// TIA Portal V20 export
FUNCTION_BLOCK "AdjLeft"   // FB525, FBD
{ S7_Optimized_Access := 'TRUE' }
// stored: AutoNumber false, MemoryReserve 100, SetENOAutomatically false
   VAR
      Var { ExternalAccessible := 'False'; ExternalVisible := 'False'; ExternalWritable := 'False'} : "TypeVar";
      Cmd { ExternalAccessible := 'False'; ExternalVisible := 'False'; ExternalWritable := 'False'} : "TypeCmd";
      Enc { ExternalAccessible := 'False'; ExternalVisible := 'False'; ExternalWritable := 'False'} : "SysCounterFast";
      Pos { ExternalAccessible := 'False'; ExternalVisible := 'False'; ExternalWritable := 'False'} : "SysPos";
      AdjSlow { ExternalAccessible := 'False'; ExternalVisible := 'False'; ExternalWritable := 'False'} : "SysMotor";
      AdjFast { ExternalAccessible := 'False'; ExternalVisible := 'False'; ExternalWritable := 'False'} : "SysLinMotC1150";
      TAutoOn { ExternalAccessible := 'False'; ExternalVisible := 'False'; ExternalWritable := 'False'} : TON_TIME;
      TAutoTarPosManOn { ExternalAccessible := 'False'; ExternalVisible := 'False'; ExternalWritable := 'False'} : TON_TIME;
      T { ExternalAccessible := 'False'; ExternalVisible := 'False'; ExternalWritable := 'False'} : Array[1..5] of IEC_TIMER;
      adjFastPnSlaveOff { ExternalAccessible := 'False'; ExternalVisible := 'False'; ExternalWritable := 'False'} : "SysPnSlaveDeactivate";
      tarOld { ExternalAccessible := 'False'; ExternalVisible := 'False'; ExternalWritable := 'False'} : DInt;
      autoTarPosMan { ExternalAccessible := 'False'; ExternalVisible := 'False'; ExternalWritable := 'False'} : Bool;
      setValueEnc { ExternalAccessible := 'False'; ExternalVisible := 'False'; ExternalWritable := 'False'} : Bool;
      autoRef { ExternalAccessible := 'False'; ExternalVisible := 'False'; ExternalWritable := 'False'} : Bool;
      posOld { ExternalAccessible := 'False'; ExternalVisible := 'False'; ExternalWritable := 'False'} : Real;
      posDiff { ExternalAccessible := 'False'; ExternalVisible := 'False'; ExternalWritable := 'False'} : Real;
   END_VAR
   VAR_TEMP
      CtrlPc : Struct
         ackErr : Bool;
         manModeActive : Bool;
         manP : Bool;
         manM : Bool;
         manRefRun : Bool;
      END_STRUCT;
      CtrlLinMot : Struct
         mode : Int;
         target : Real;
         acc : Real;
         dec : Real;
         jerk : Real;
         speed : Real;
      END_STRUCT;
      refPosDiff : DInt;
      offsetNoStd : Real;
      refPosDiffCalib : DInt;
      modeCalib : Int;
      disMechanicToZero : Int;   // distance mechanic part left to zero [mm]
   END_VAR
   VAR_TEMP   // added for the SCL form of the ladder/FBD networks
      _w1 : Bool;
   END_VAR
BEGIN

REGION Network 1 (SCL): offset for no standard calibration
   (* 
   normally the distance from camera TO board should be 550mm
   for special application the distance is different
   the distance can be changed in the goldeneye program
   if its different then 550mm a offset will be added
   *)
   #offsetNoStd := 0.0;
   IF "ComRd".Data.Left.RefPosToBoard <> 550 THEN
       #offsetNoStd := (DINT_TO_REAL("ComRd".Data.Left.RefPosToBoard) - 550.0);
   ELSE
       #offsetNoStd := 0.0;
   END_IF;
END_REGION

REGION Network 2 (SCL): calibration value for offset
   (* 
   modus for calibartion
   camera must be referenced first
   mode 1 -->   the camera must be moved manually to position 550mm from board and
                 then press "Set Nullpoint"
   mode 2 -->   the camera must be moved to a other position and
                 then must be measured from the calibration tool to the camera and
                 this value must be putted in after pressing "Set Nullpoint"
   *)     
   #disMechanicToZero := 870;  
   #modeCalib := 2;
   IF #modeCalib = 1 THEN
       #refPosDiffCalib := "ComRd".Data.Left.TargetPos;
   ELSIF #modeCalib = 2 THEN
       #refPosDiffCalib := (#disMechanicToZero * 10) - ("ComRd".Data.Left.CalibratePos + 5500);
   END_IF;
END_REGION

REGION Network 3 (SCL): calibration value from pc
   "ComSd".Data.Left.SetCalibratePosOk := FALSE;

   IF "ComRd".Data.Left.SetCalibratePos THEN

       IF "G".Cfg.adjLeftActive THEN
           #refPosDiff := REAL_TO_DINT("Enc"."8BC1.L".act * 10.0) - #refPosDiffCalib;
       ELSIF "G".Cfg.adjLeftActiveLinMot THEN
           #refPosDiff := REAL_TO_DINT("Enc"."8U1.L".act * 10.0) - #refPosDiffCalib;
       END_IF;

       "Ref".adjLeftCalOffset := #refPosDiff;
       "ComSd".Data.Left.SetCalibratePosOk := TRUE;

   END_IF;
END_REGION

REGION Network 4 (SCL): target position
   #Cmd.target := "G".Batch.width / 2.0;
   IF "G".Cfg.modeBoardPassing = 2 AND ("G".Cfg.modeDimension = 2 OR "G".Cfg.modeDimension = 4) AND NOT "G".Batch.stdActive THEN
       #Cmd.target := "G".Batch.width / 2.0 + ("G".Batch.widthMeasure - "G".Batch.width);
   END_IF;

   IF "G".Cfg.modeBoardPassing = 3 AND ("G".Cfg.modeDimension = 2 OR "G".Cfg.modeDimension = 4) AND NOT "G".Batch.stdActive THEN
       #Cmd.target := "G".Batch.senLeftVal;
   END_IF;

   IF #autoTarPosMan THEN
       #Cmd.target := DINT_TO_REAL(("ComRd".Data.Left.TargetPos)) / 10.0;
   END_IF;

   "Ref".adjLeftTar := #Cmd.target + (DINT_TO_REAL("Ref".adjLeftCalOffset) / 10.0) + #offsetNoStd + "Enc"."8B1.B".offset;
END_REGION

REGION Network 5 (SCL): data from pc
   IF NOT "G".errComPc THEN
       #CtrlPc.manModeActive := "ComRd".Data.Left.ManModeActive;
       #CtrlPc.manP := "ComRd".Data.Left.ManPlus;
       #CtrlPc.manM := "ComRd".Data.Left.ManMinus;
       #CtrlPc.manRefRun := "ComRd".Data.Left.ManRefRun;
   ELSE
       #CtrlPc.manModeActive := TRUE;
       #CtrlPc.manP := FALSE;
       #CtrlPc.manM := FALSE;
       #CtrlPc.manRefRun := FALSE;
   END_IF;
   #CtrlPc.ackErr := "G".ack;
END_REGION

REGION Network 6: off
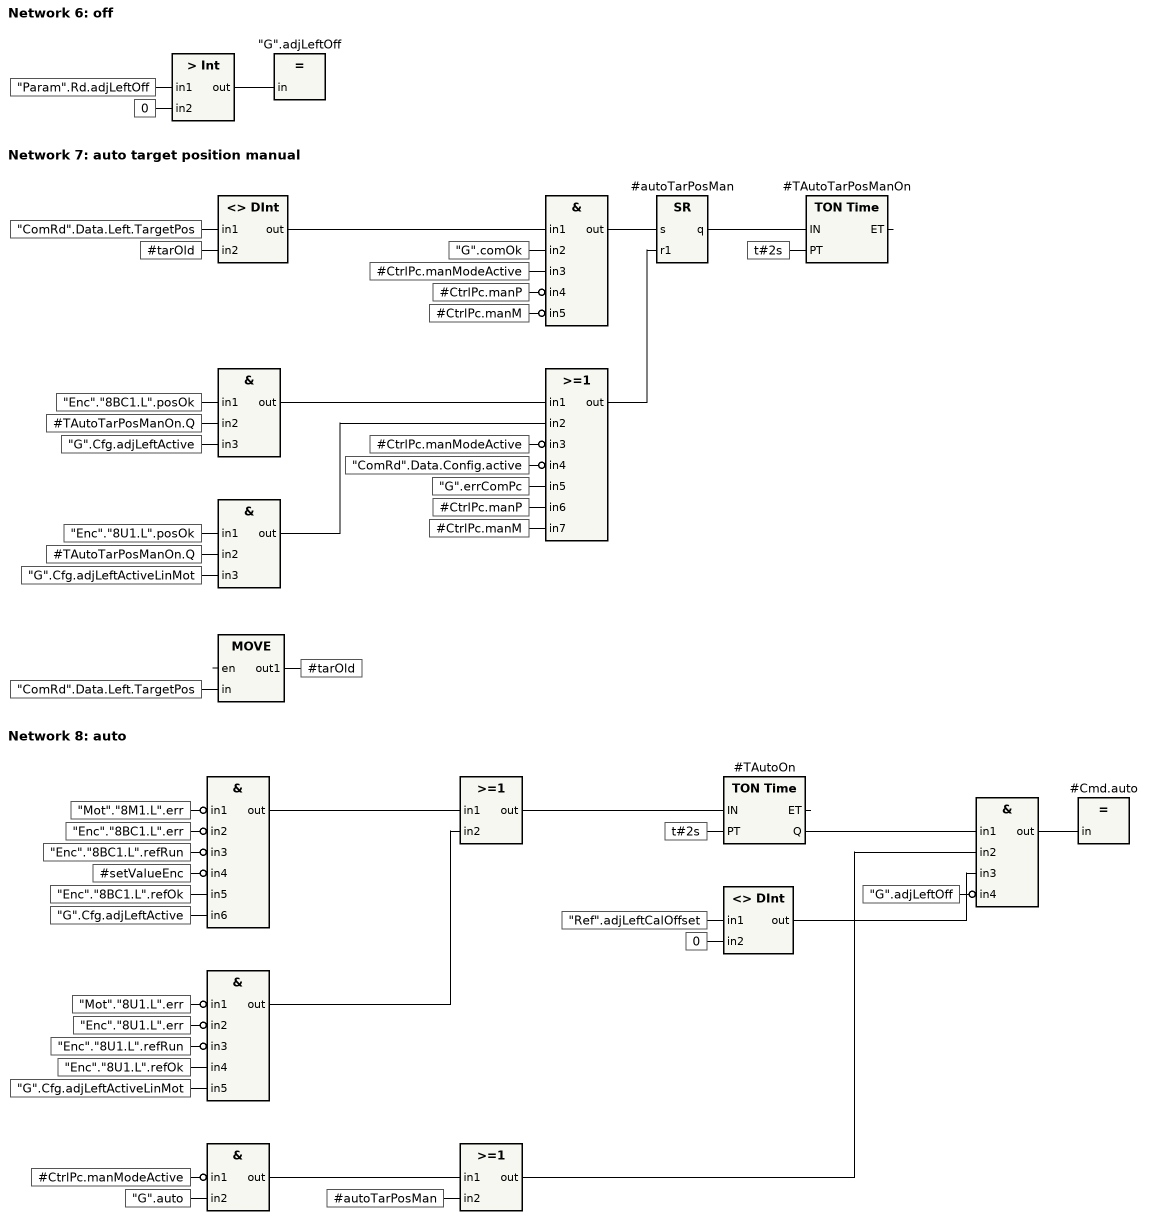
   "G".adjLeftOff := "Param".Rd.adjLeftOff > 0;
END_REGION

REGION Network 7: auto target position manual
   IF ("ComRd".Data.Left.TargetPos <> #tarOld) AND "G".comOk AND #CtrlPc.manModeActive AND NOT #CtrlPc.manP AND NOT #CtrlPc.manM THEN
       #autoTarPosMan := TRUE;   // SR flip-flop
   END_IF;
   IF ("Enc"."8BC1.L".posOk AND #TAutoTarPosManOn.Q AND "G".Cfg.adjLeftActive) OR ("Enc"."8U1.L".posOk AND #TAutoTarPosManOn.Q AND "G".Cfg.adjLeftActiveLinMot) OR NOT #CtrlPc.manModeActive OR NOT "ComRd".Data.Config.active OR "G".errComPc OR #CtrlPc.manP OR #CtrlPc.manM THEN
       #autoTarPosMan := FALSE;
   END_IF;
   #TAutoTarPosManOn(IN := #autoTarPosMan, PT := t#2s);   // TON
   #tarOld := "ComRd".Data.Left.TargetPos;
END_REGION

REGION Network 8: auto
   #TAutoOn(IN := (NOT "Mot"."8M1.L".err AND NOT "Enc"."8BC1.L".err AND NOT "Enc"."8BC1.L".refRun AND NOT #setValueEnc AND "Enc"."8BC1.L".refOk AND "G".Cfg.adjLeftActive) OR (NOT "Mot"."8U1.L".err AND NOT "Enc"."8U1.L".err AND NOT "Enc"."8U1.L".refRun AND "Enc"."8U1.L".refOk AND "G".Cfg.adjLeftActiveLinMot),   // TON
            PT := t#2s);
   #Cmd.auto := #TAutoOn.Q AND ((NOT #CtrlPc.manModeActive AND "G".auto) OR #autoTarPosMan) AND ("Ref".adjLeftCalOffset <> 0) AND NOT "G".adjLeftOff;
END_REGION

REGION Network 9: manual
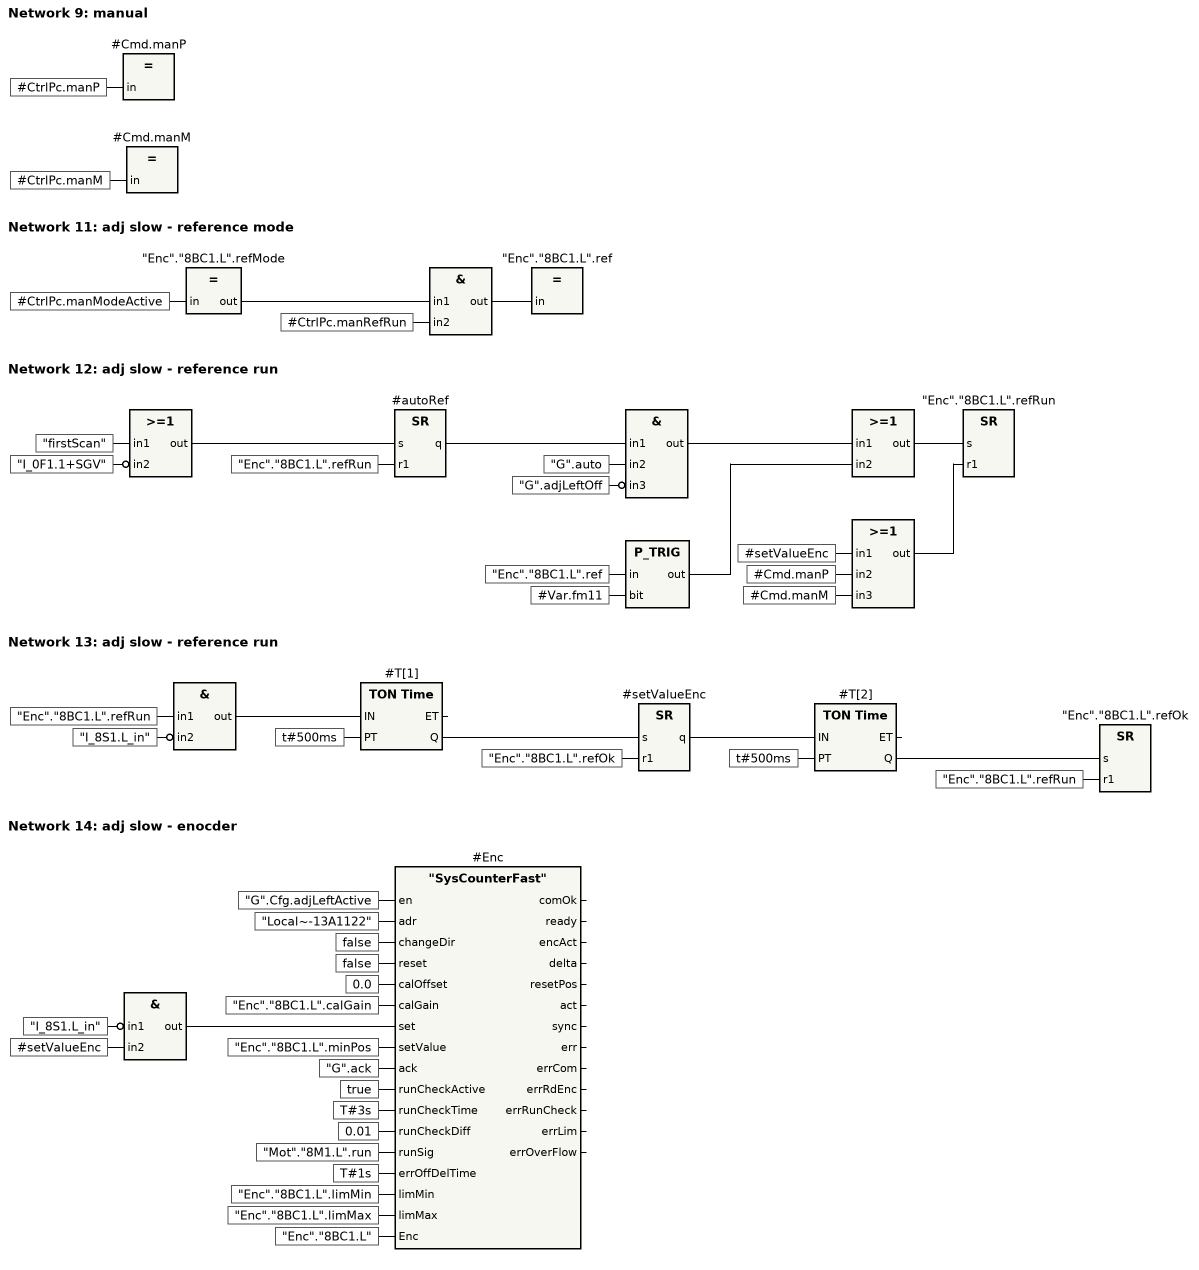
   #Cmd.manP := #CtrlPc.manP;
   #Cmd.manM := #CtrlPc.manM;
END_REGION

REGION Network 10 (SCL): adj slow - calibration value
   "Enc"."8BC1.L".calGain := -0.0275;

   "Enc"."8BC1.L".minPos := 10.0;
   "Enc"."8BC1.L".maxPos := 210.0;

   "Enc"."8BC1.L".limMin := "Enc"."8BC1.L".minPos - 5.0;
   "Enc"."8BC1.L".limMax := "Enc"."8BC1.L".maxPos + 5.0;

   "Enc"."8BC1.L".tarMinPos := "Enc"."8BC1.L".minPos + 0.0;
   "Enc"."8BC1.L".tarMaxPos := "Enc"."8BC1.L".maxPos - 0.0;
END_REGION

REGION Network 11: adj slow - reference mode
   "Enc"."8BC1.L".refMode := #CtrlPc.manModeActive;
   "Enc"."8BC1.L".ref := #CtrlPc.manModeActive AND #CtrlPc.manRefRun;
END_REGION

REGION Network 12: adj slow - reference run
   IF "firstScan" OR NOT "I_0F1.1+SGV" THEN
       #autoRef := TRUE;   // SR flip-flop
   END_IF;
   IF "Enc"."8BC1.L".refRun THEN #autoRef := FALSE; END_IF;
   #_w1 := "Enc"."8BC1.L".ref AND NOT #Var.fm11;   // rising edge
   #Var.fm11 := "Enc"."8BC1.L".ref;
   IF (#autoRef AND "G".auto AND NOT "G".adjLeftOff) OR #_w1 THEN
       "Enc"."8BC1.L".refRun := TRUE;   // SR flip-flop
   END_IF;
   IF #setValueEnc OR #Cmd.manP OR #Cmd.manM THEN "Enc"."8BC1.L".refRun := FALSE; END_IF;
END_REGION

REGION Network 13: adj slow - reference run
   #T[1].TON(IN := "Enc"."8BC1.L".refRun AND NOT "I_8S1.L_in", PT := t#500ms);
   IF #T[1].Q THEN
       #setValueEnc := TRUE;   // SR flip-flop
   END_IF;
   IF "Enc"."8BC1.L".refOk THEN #setValueEnc := FALSE; END_IF;
   #T[2].TON(IN := #setValueEnc, PT := t#500ms);
   IF #T[2].Q THEN
       "Enc"."8BC1.L".refOk := TRUE;   // SR flip-flop
   END_IF;
   IF "Enc"."8BC1.L".refRun THEN "Enc"."8BC1.L".refOk := FALSE; END_IF;
END_REGION

REGION Network 14: adj slow - enocder
   IF "G".Cfg.adjLeftActive THEN
       #Enc(adr := "Local~-13A1122",   // "SysCounterFast"
            changeDir := false,
            reset := false,
            calOffset := 0.0,
            calGain := "Enc"."8BC1.L".calGain,
            set := NOT "I_8S1.L_in" AND #setValueEnc,
            setValue := "Enc"."8BC1.L".minPos,
            ack := "G".ack,
            runCheckActive := true,
            runCheckTime := T#3s,
            runCheckDiff := 0.01,
            runSig := "Mot"."8M1.L".run,
            errOffDelTime := T#1s,
            limMin := "Enc"."8BC1.L".limMin,
            limMax := "Enc"."8BC1.L".limMax,
            Enc := "Enc"."8BC1.L");
   END_IF;
END_REGION

REGION Network 15: adj slow - pos
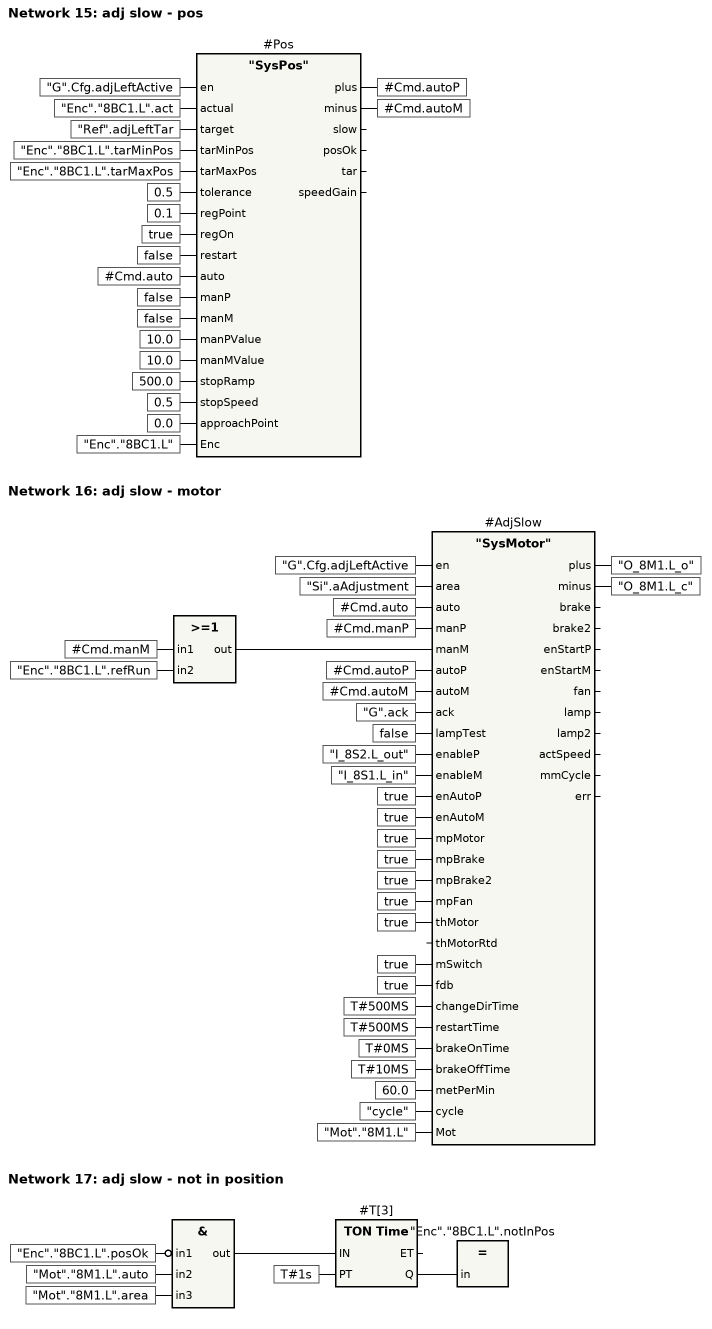
   IF "G".Cfg.adjLeftActive THEN
       #Pos(actual := "Enc"."8BC1.L".act,   // "SysPos"
            target := "Ref".adjLeftTar,
            tarMinPos := "Enc"."8BC1.L".tarMinPos,
            tarMaxPos := "Enc"."8BC1.L".tarMaxPos,
            tolerance := 0.5,
            regPoint := 0.1,
            regOn := true,
            restart := false,
            auto := #Cmd.auto,
            manP := false,
            manM := false,
            manPValue := 10.0,
            manMValue := 10.0,
            stopRamp := 500.0,
            stopSpeed := 0.5,
            approachPoint := 0.0,
            Enc := "Enc"."8BC1.L",
            plus => #Cmd.autoP,
            minus => #Cmd.autoM);
   END_IF;
END_REGION

REGION Network 16: adj slow - motor
   IF "G".Cfg.adjLeftActive THEN
       #AdjSlow(area := "Si".aAdjustment,   // "SysMotor"
                auto := #Cmd.auto,
                manP := #Cmd.manP,
                manM := #Cmd.manM OR "Enc"."8BC1.L".refRun,
                autoP := #Cmd.autoP,
                autoM := #Cmd.autoM,
                ack := "G".ack,
                lampTest := false,
                enableP := "I_8S2.L_out",
                enableM := "I_8S1.L_in",
                enAutoP := true,
                enAutoM := true,
                mpMotor := true,
                mpBrake := true,
                mpBrake2 := true,
                mpFan := true,
                thMotor := true,
                mSwitch := true,
                fdb := true,
                changeDirTime := T#500MS,
                restartTime := T#500MS,
                brakeOnTime := T#0MS,
                brakeOffTime := T#10MS,
                metPerMin := 60.0,
                cycle := "cycle",
                Mot := "Mot"."8M1.L",
                plus => "O_8M1.L_o",
                minus => "O_8M1.L_c");
   END_IF;
END_REGION

REGION Network 17: adj slow - not in position
   #T[3].TON(IN := NOT "Enc"."8BC1.L".posOk AND "Mot"."8M1.L".auto AND "Mot"."8M1.L".area, PT := T#1s);
   "Enc"."8BC1.L".notInPos := #T[3].Q;
END_REGION

REGION Network 18: adj slow - sensor monitoring
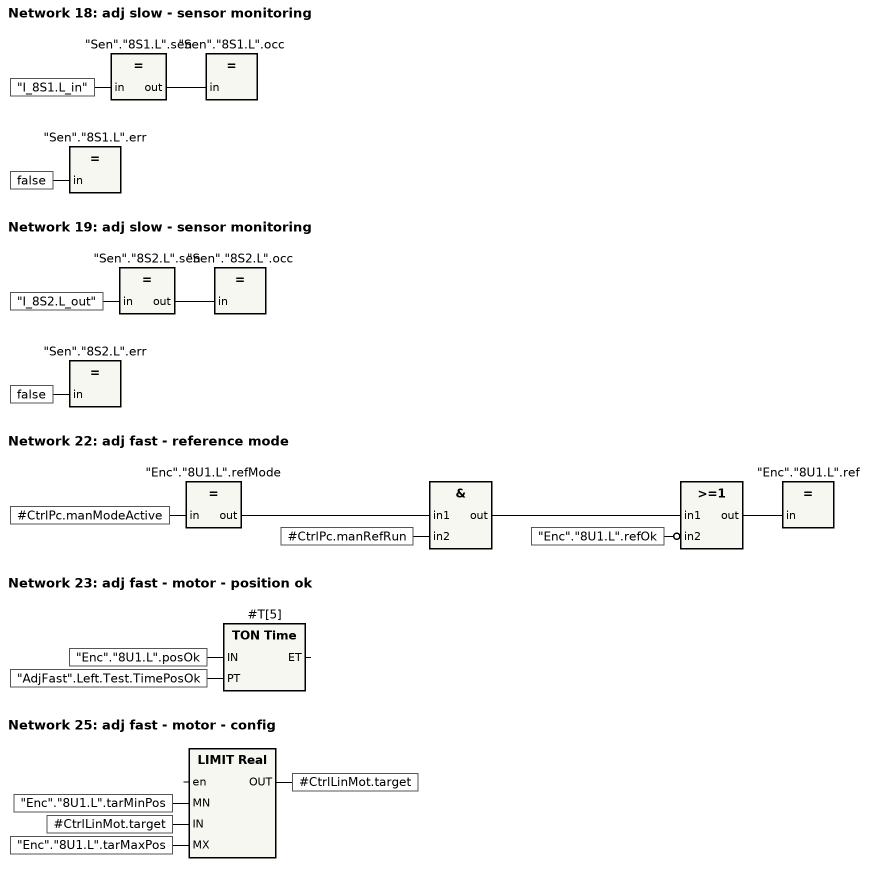
   "Sen"."8S1.L".sen := "I_8S1.L_in";
   "Sen"."8S1.L".occ := "I_8S1.L_in";
   "Sen"."8S1.L".err := false;
END_REGION

REGION Network 19: adj slow - sensor monitoring
   "Sen"."8S2.L".sen := "I_8S2.L_out";
   "Sen"."8S2.L".occ := "I_8S2.L_out";
   "Sen"."8S2.L".err := false;
END_REGION

REGION Network 21 (SCL): adj fast - calibration value
   "Enc"."8U1.L".calGain := 1.0;

   "Enc"."8U1.L".minPos := 5.0;
   "Enc"."8U1.L".maxPos := 155.0;

   "Enc"."8U1.L".limMin := "Enc"."8U1.L".minPos - 5.0;
   "Enc"."8U1.L".limMax := "Enc"."8U1.L".maxPos + 5.0;

   "Enc"."8U1.L".tarMinPos := "Enc"."8U1.L".minPos + 0.0;
   "Enc"."8U1.L".tarMaxPos := "Enc"."8U1.L".maxPos - 0.0;
END_REGION

REGION Network 22: adj fast - reference mode
   "Enc"."8U1.L".refMode := #CtrlPc.manModeActive;
   "Enc"."8U1.L".ref := (#CtrlPc.manModeActive AND #CtrlPc.manRefRun) OR NOT "Enc"."8U1.L".refOk;
END_REGION

REGION Network 23: adj fast - motor - position ok
   #T[5].TON(IN := "Enc"."8U1.L".posOk, PT := "AdjFast".Left.Test.TimePosOk);
END_REGION

REGION Network 24 (SCL): adj fast - motor - config

   //############################################################
   // min            5     mm
   // max          155     mm

   // speed        02      m/s
   // acc/dec      24      m/s2
   // jerk         450     m/s3

   // mode         BestehornVAJ
   //############################################################

   // only testmode for plc
   IF "AdjFast".Left.Test.ModeActive AND NOT #CtrlPc.manModeActive THEN
       IF "AdjFast".Left.Test.TarPos = "AdjFast".Left.Test.TarPos1 AND #T[5].Q THEN
           "AdjFast".Left.Test.TarPos := "AdjFast".Left.Test.TarPos2;
       ELSIF "AdjFast".Left.Test.TarPos = "AdjFast".Left.Test.TarPos2 AND #T[5].Q THEN
           "AdjFast".Left.Test.TarPos := "AdjFast".Left.Test.TarPos1;
       END_IF;
       "Ref".adjLeftTar := "AdjFast".Left.Test.TarPos;
   END_IF;

   // active mode
   #CtrlLinMot.mode := 3;
   #CtrlLinMot.target := "Ref".adjLeftTar;
   #CtrlLinMot.speed := 2.0;
   #CtrlLinMot.acc := 24.0;
   #CtrlLinMot.dec := 0.0;
   #CtrlLinMot.jerk := 450.0;

   // only testmode for plc
   IF "AdjFast".Left.Mode = 1 THEN
       #CtrlLinMot.mode := 1;
       #CtrlLinMot.target := "AdjFast".Left.VAI.Par1;
       #CtrlLinMot.speed := "AdjFast".Left.VAI.Par2;
       #CtrlLinMot.acc := "AdjFast".Left.VAI.Par3;
       #CtrlLinMot.dec := "AdjFast".Left.VAI.Par4;
       #CtrlLinMot.jerk := 0.0;
   ELSIF "AdjFast".Left.Mode = 2 THEN
       #CtrlLinMot.mode := 2;
       #CtrlLinMot.target := "AdjFast".Left.SinVA.Par1;
       #CtrlLinMot.speed := "AdjFast".Left.SinVA.Par2;
       #CtrlLinMot.acc := "AdjFast".Left.SinVA.Par3;
       #CtrlLinMot.dec := 0.0;
       #CtrlLinMot.jerk := 0.0;
   ELSIF "AdjFast".Left.Mode = 3 THEN
       #CtrlLinMot.mode := 3;
       #CtrlLinMot.target := "AdjFast".Left.BestehornVAJ.Par1;
       #CtrlLinMot.speed := "AdjFast".Left.BestehornVAJ.Par2;
       #CtrlLinMot.acc := "AdjFast".Left.BestehornVAJ.Par3;
       #CtrlLinMot.dec := 0.0;
       #CtrlLinMot.jerk := "AdjFast".Left.BestehornVAJ.Par4;
   END_IF;
END_REGION

REGION Network 25: adj fast - motor - config
   #CtrlLinMot.target := LIMIT(MN := "Enc"."8U1.L".tarMinPos, IN := #CtrlLinMot.target, MX := "Enc"."8U1.L".tarMaxPos);
END_REGION

REGION Network 26: adj fast - motor
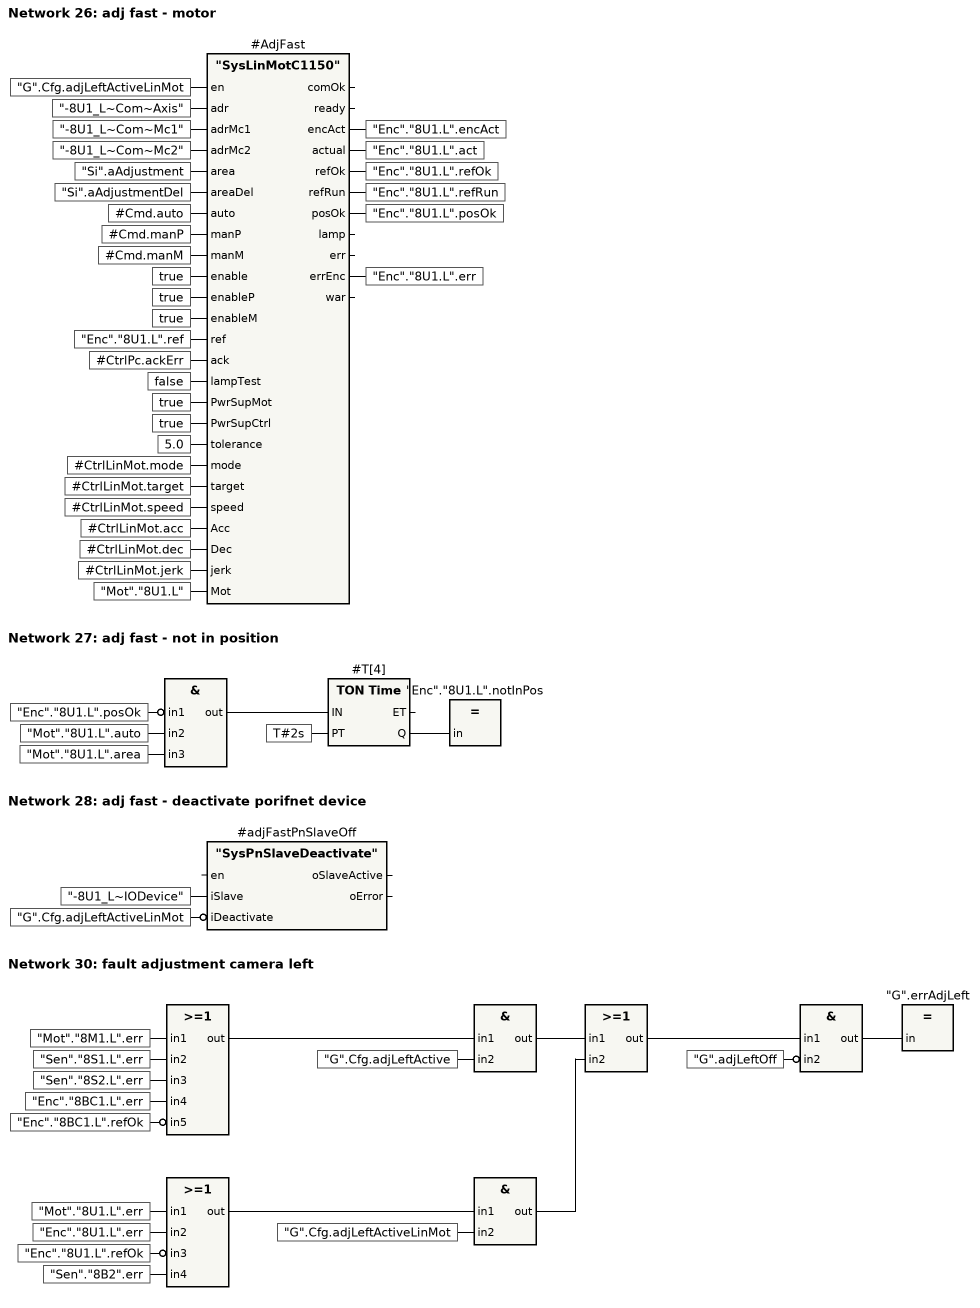
   IF "G".Cfg.adjLeftActiveLinMot THEN
       #AdjFast(adr := "-8U1_L~Com~Axis",   // "SysLinMotC1150"
                adrMc1 := "-8U1_L~Com~Mc1",
                adrMc2 := "-8U1_L~Com~Mc2",
                area := "Si".aAdjustment,
                areaDel := "Si".aAdjustmentDel,
                auto := #Cmd.auto,
                manP := #Cmd.manP,
                manM := #Cmd.manM,
                enable := true,
                enableP := true,
                enableM := true,
                ref := "Enc"."8U1.L".ref,
                ack := #CtrlPc.ackErr,
                lampTest := false,
                PwrSupMot := true,
                PwrSupCtrl := true,
                tolerance := 5.0,
                mode := #CtrlLinMot.mode,
                target := #CtrlLinMot.target,
                speed := #CtrlLinMot.speed,
                Acc := #CtrlLinMot.acc,
                Dec := #CtrlLinMot.dec,
                jerk := #CtrlLinMot.jerk,
                Mot := "Mot"."8U1.L",
                encAct => "Enc"."8U1.L".encAct,
                actual => "Enc"."8U1.L".act,
                refOk => "Enc"."8U1.L".refOk,
                refRun => "Enc"."8U1.L".refRun,
                posOk => "Enc"."8U1.L".posOk,
                errEnc => "Enc"."8U1.L".err);
   END_IF;
END_REGION

REGION Network 27: adj fast - not in position
   #T[4].TON(IN := NOT "Enc"."8U1.L".posOk AND "Mot"."8U1.L".auto AND "Mot"."8U1.L".area, PT := T#2s);
   "Enc"."8U1.L".notInPos := #T[4].Q;
END_REGION

REGION Network 28: adj fast - deactivate porifnet device
   #adjFastPnSlaveOff(iSlave := "-8U1_L~IODevice", iDeactivate := NOT "G".Cfg.adjLeftActiveLinMot);   // "SysPnSlaveDeactivate"
END_REGION

REGION Network 30: fault adjustment camera left
   "G".errAdjLeft := ((("Mot"."8M1.L".err OR "Sen"."8S1.L".err OR "Sen"."8S2.L".err OR "Enc"."8BC1.L".err OR NOT "Enc"."8BC1.L".refOk) AND "G".Cfg.adjLeftActive) OR (("Mot"."8U1.L".err OR "Enc"."8U1.L".err OR NOT "Enc"."8U1.L".refOk OR "Sen"."8B2".err) AND "G".Cfg.adjLeftActiveLinMot)) AND NOT "G".adjLeftOff;
END_REGION

REGION Network 31 (SCL): data to pc
   IF "G".Cfg.adjLeftActive THEN
       "Ref".adjLeftAct := REAL_TO_DINT("Enc"."8BC1.L".act * 10.0) - "Ref".adjLeftCalOffset - REAL_TO_DINT(#offsetNoStd * 10.0);
       "ComSd".Data.Left.ActualEncPos := REAL_TO_DINT("Enc"."8BC1.L".act * 10.0);
       "ComSd".Data.Left.ActualPos :=  "Ref".adjLeftAct;
       "ComSd".Data.Left.LimitSwitchMin := "Sen"."8S1.L".sen;
       "ComSd".Data.Left.LimitSwitchMax := "Sen"."8S2.L".sen;
       "ComSd".Data.Left.Err := "Mot"."8M1.L".err;
       "ComSd".Data.Left.ErrEnc := "Enc"."8BC1.L".err;
       "ComSd".Data.Left.PosOk := "Enc"."8BC1.L".posOk;
       "ComSd".Data.Left.Plus := "Mot"."8M1.L".plus;
       "ComSd".Data.Left.Minus := "Mot"."8M1.L".minus;
       "ComSd".Data.Left.refRun := "Enc"."8BC1.L".refRun;
       "ComSd".Data.Left.refOk := "Enc"."8BC1.L".refOk;
   ELSIF  "G".Cfg.adjLeftActiveLinMot THEN
       "Ref".adjLeftAct := REAL_TO_DINT("Enc"."8U1.L".act * 10.0) - "Ref".adjLeftCalOffset - REAL_TO_DINT(#offsetNoStd * 10.0);
       "ComSd".Data.Left.ActualEncPos := REAL_TO_DINT("Enc"."8U1.L".act * 10.0);
       "ComSd".Data.Left.ActualPos :=  "Ref".adjLeftAct;
       "ComSd".Data.Left.LimitSwitchMin := TRUE;
       "ComSd".Data.Left.LimitSwitchMax := TRUE;
       "ComSd".Data.Left.Err := "Mot"."8U1.L".err;
       "ComSd".Data.Left.ErrEnc := "Enc"."8U1.L".err;
       "ComSd".Data.Left.PosOk := "Enc"."8U1.L".posOk;
       "ComSd".Data.Left.Plus := "Mot"."8U1.L".plus;
       "ComSd".Data.Left.Minus := "Mot"."8U1.L".minus;
       "ComSd".Data.Left.refRun := "Enc"."8U1.L".refRun;
       "ComSd".Data.Left.refOk := "Enc"."8U1.L".refOk;
   ELSE
       "ComSd".Data.Left.ActualEncPos := 0;
       "ComSd".Data.Left.ActualPos := 0;
       "ComSd".Data.Left.LimitSwitchMin := FALSE;
       "ComSd".Data.Left.LimitSwitchMax := FALSE;
       "ComSd".Data.Left.Err := FALSE;
       "ComSd".Data.Left.ErrEnc := FALSE;
       "ComSd".Data.Left.PosOk := True;
       "ComSd".Data.Left.Plus := FALSE;
       "ComSd".Data.Left.Minus := FALSE;
       "ComSd".Data.Left.refRun := FALSE;
       "ComSd".Data.Left.refOk := TRUE;
   END_IF;
END_REGION

REGION Network 32: current monitoring - auto
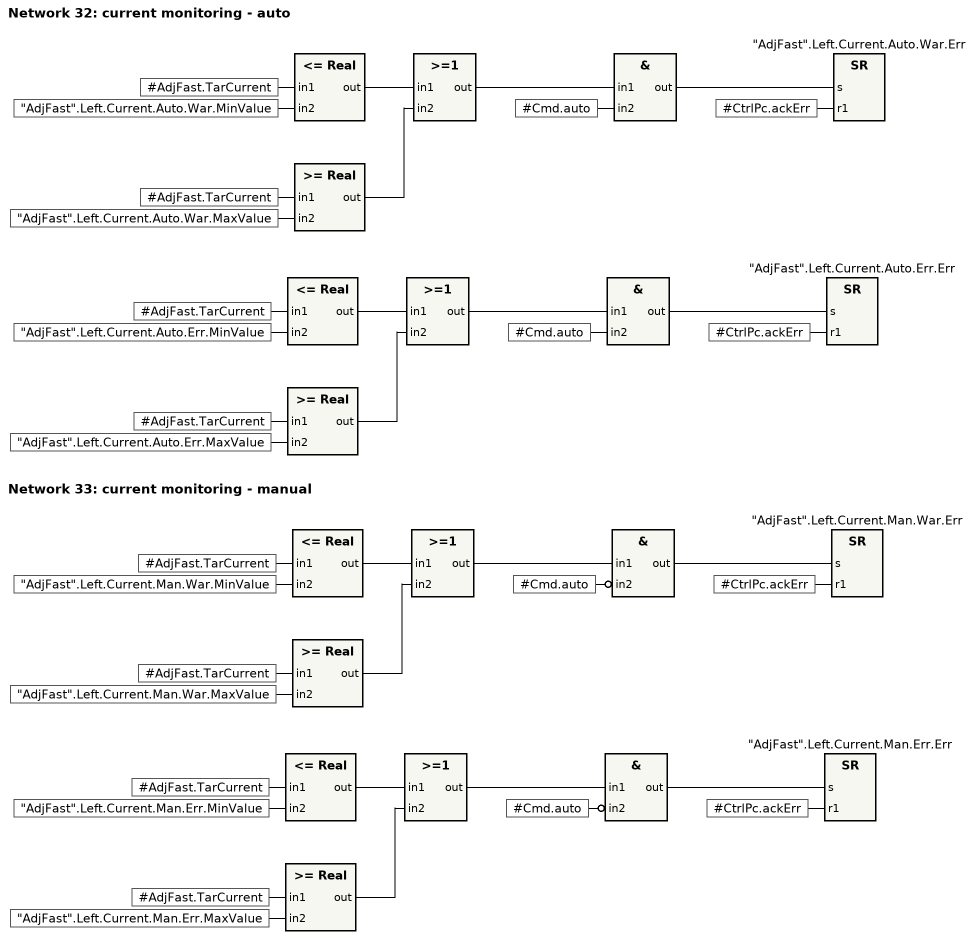
   IF ((#AdjFast.TarCurrent <= "AdjFast".Left.Current.Auto.War.MinValue) OR (#AdjFast.TarCurrent >= "AdjFast".Left.Current.Auto.War.MaxValue)) AND #Cmd.auto THEN
       "AdjFast".Left.Current.Auto.War.Err := TRUE;   // SR flip-flop
   END_IF;
   IF #CtrlPc.ackErr THEN "AdjFast".Left.Current.Auto.War.Err := FALSE; END_IF;
   IF ((#AdjFast.TarCurrent <= "AdjFast".Left.Current.Auto.Err.MinValue) OR (#AdjFast.TarCurrent >= "AdjFast".Left.Current.Auto.Err.MaxValue)) AND #Cmd.auto THEN
       "AdjFast".Left.Current.Auto.Err.Err := TRUE;   // SR flip-flop
   END_IF;
   IF #CtrlPc.ackErr THEN "AdjFast".Left.Current.Auto.Err.Err := FALSE; END_IF;
END_REGION

REGION Network 33: current monitoring - manual
   IF ((#AdjFast.TarCurrent <= "AdjFast".Left.Current.Man.War.MinValue) OR (#AdjFast.TarCurrent >= "AdjFast".Left.Current.Man.War.MaxValue)) AND NOT #Cmd.auto THEN
       "AdjFast".Left.Current.Man.War.Err := TRUE;   // SR flip-flop
   END_IF;
   IF #CtrlPc.ackErr THEN "AdjFast".Left.Current.Man.War.Err := FALSE; END_IF;
   IF ((#AdjFast.TarCurrent <= "AdjFast".Left.Current.Man.Err.MinValue) OR (#AdjFast.TarCurrent >= "AdjFast".Left.Current.Man.Err.MaxValue)) AND NOT #Cmd.auto THEN
       "AdjFast".Left.Current.Man.Err.Err := TRUE;   // SR flip-flop
   END_IF;
   IF #CtrlPc.ackErr THEN "AdjFast".Left.Current.Man.Err.Err := FALSE; END_IF;
END_REGION
END_FUNCTION_BLOCK
